(*
SPDX-FileCopyrightText: © 2026 Oleksandr Tiutyk <trofimich@gmail.com>
SPDX-License-Identifier: MIT
License: https://opensource.org/license/mit
*)

//!<param name="POSITIVE_INFINITY">IEEE 754 +Infinity</param>

//!<param name="NEGATIVE_INFINITY">IEEE 754 -Infinity</param>

{attribute 'no_explicit_call' := 'do not call this function block directly'} 
PROGRAM Reals
VAR CONSTANT
	MIN_VALUE : REAL := -3.402823E+38;
	MAX_VALUE : REAL := +3.402823E+38;
	
    POSITIVE_INFINITY : REAL_UNION := (Raw := 16#7F800000); 
    NEGATIVE_INFINITY : REAL_UNION := (Raw := 16#FF800000); 
    NOT_A_NUMBER : REAL := TO_REAL(LOG(-1)); // REAL_UNION := (Raw := 16#7FC00000); // IEEE 754 NaN	
END_VAR
VAR
	{attribute 'hide'} 
	_ClassName : STRING := __POUNAME();
END_VAR

{attribute 'monitoring' := 'call'}
PROPERTY ClassName : REFERENCE TO STRING
GET
ClassName REF= _ClassName;
END_GET
END_PROPERTY

{attribute 'monitoring' := 'call'}
PROPERTY NamespaceName : REFERENCE TO STRING
GET
NamespaceName REF= CurrentNamespace.Name;
END_GET
END_PROPERTY

END_PROGRAM

(* stored: Version 1.1.0.1
   POU Reals: Id {361c062a-943b-4db7-ab4a-7715ff446a31}, SpecialFunc None
   Property ClassName: Id {9df65ee2-61ad-4aa6-8540-da6369d277dd}
   Get Get: Id {f3e499ff-278e-4944-9b5a-c3c32eaeeaeb}
   Property NamespaceName: Id {38bfc198-2daa-457d-8569-d0dd6eafc0d0}
   Get Get: Id {f423181e-b835-486d-a0e9-cbf1e9bf75ba} *)
